FUNCTION_BLOCK FB_DigitalSensor IMPLEMENTS I_DigitalSensor
VAR_INPUT
    // The physical hardware terminal mapping
    bRawInput AT %I* : BOOL; 
    
    // NEW: HiL Simulation Hooks
    bSimulationMode  : BOOL; // TRUE = Ignore physical %I*, use bSimulationInput
    {attribute 'TcLinkTo' := '1'}
	bSimulationInput AT %I* : BOOL;
END_VAR
VAR
    // Internal State (Private)
    bActive         : BOOL;
    bEffectiveInput : BOOL; // Multiplexer output
    bInvert         : BOOL;
    
    // Edge Detection
    fbRisingEdge  : R_TRIG;
    fbFallingEdge : F_TRIG;
END_VAR

// =========================================================
// 1. HARDWARE VS. SIMULATION MULTIPLEXER
// =========================================================
IF bSimulationMode THEN
    bEffectiveInput := bSimulationInput; // Listen to Python Twin
ELSE
    bEffectiveInput := bRawInput;        // Listen to Physical IO Terminal
END_IF

// =========================================================
// 2. Handle Wiring Logic (Normally Open vs Normally Closed)
// =========================================================
IF bInvert THEN
    bActive := NOT bEffectiveInput;
ELSE
    bActive := bEffectiveInput;
END_IF

// =========================================================
// 3. Run the Edge Detection Blocks
// =========================================================
fbRisingEdge(CLK := bActive);
fbFallingEdge(CLK := bActive);

PROPERTY P_FallingEdge : BOOL
GET
P_FallingEdge := fbFallingEdge.Q;
END_GET
END_PROPERTY

PROPERTY P_InvertLogic : BOOL
GET
P_InvertLogic := bInvert;
END_GET
SET
bInvert := P_InvertLogic;
END_SET
END_PROPERTY

PROPERTY P_IsActive : BOOL
GET
P_IsActive := bActive;
END_GET
END_PROPERTY

PROPERTY P_RawInput : BOOL
GET
P_RawInput := bRawInput;
END_GET
SET
bRawInput := P_RawInput;
END_SET
END_PROPERTY

PROPERTY P_RisingEdge : BOOL
GET
P_RisingEdge := fbRisingEdge.Q;
END_GET
END_PROPERTY

END_FUNCTION_BLOCK

(* stored: Version 1.1.0.1
   POU FB_DigitalSensor: Id {6a39500a-bba7-4420-a58b-3b1e1df2d295}, SpecialFunc None
   Property P_FallingEdge: Id {72f4abad-3ae3-4f58-b135-9f5a75a1fd1b}
   Get Get: Id {b0ae2ae5-df28-4956-9e04-dca118232247}
   Property P_InvertLogic: Id {57b94ec5-d24f-4c9c-a6b7-07a035eda686}
   Get Get: Id {20e957c8-a18e-4390-a9c2-49240c515bf6}
   Set Set: Id {c82c233e-2a1a-4b38-a570-354712badd9a}
   Property P_IsActive: Id {6658c044-a2a4-4549-af8e-3f2dbece7dd9}
   Get Get: Id {e4a1d8ae-496f-4623-8545-04bb1bf31e3c}
   Property P_RawInput: Id {1888c39b-44a9-4695-9d1c-9125368feed5}
   Get Get: Id {b87ac34c-a466-45f9-9db9-d1c61bf882ca}
   Set Set: Id {ef2d70ca-93e8-45c7-890a-8f169738602f}
   Property P_RisingEdge: Id {1f8356ea-8544-48ad-887b-04c9041b4561}
   Get Get: Id {89600acc-e52f-4c87-ad9e-f13342bf3b69} *)
